{attribute 'qualified_only'}
VAR_GLOBAL
		EtherCAT_Master_Duplicates : EtherCAT_Master_Duplicates_CB89F35C;
END_VAR

(* stored: Version 1.2.0.0, ProductVersion 3.1.4024.9
   GVL GVL_iXlinker: Id {eb6a60fb-f800-4891-a346-7f3c31aa48c6} *)
